TYPE FILE_SERVER_DATA :
STRUCT
	FILE_OPEN : BOOL;
	FILENAME : STRING;
	MODE : BYTE;
	OFFSET : UDINT;
	FILE_SIZE : UDINT;
	AUTO_CLOSE : TIME;
	ERROR : BYTE;
END_STRUCT
END_TYPE

(* stored: Version 1.1.0.1, ProductVersion 3.1.4022.7
   DUT FILE_SERVER_DATA: Id {2b1e8820-4a50-4601-97c6-7d087efa33b4} *)
